FUNCTION_BLOCK Robot_Task_CAT (* Composite Function Block Type *)
  (* Standard: 61499-2 *)
  (* Version 0.0, 10/8/2025, Schneider Electric, template *)
  PACKAGE Main;
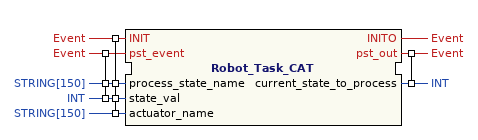
  EVENT_INPUT
    INIT WITH process_state_name, state_val, actuator_name; (* Initialization Request *)
    pst_event WITH process_state_name, state_val;
  END_EVENT
  EVENT_OUTPUT
    INITO; (* Initialization Confirm *)
    pst_out WITH current_state_to_process;
  END_EVENT
  VAR_INPUT
    process_state_name : STRING[150];
    state_val : INT;
    actuator_name : STRING[150];
  END_VAR
  VAR_OUTPUT
    current_state_to_process : INT;
  END_VAR
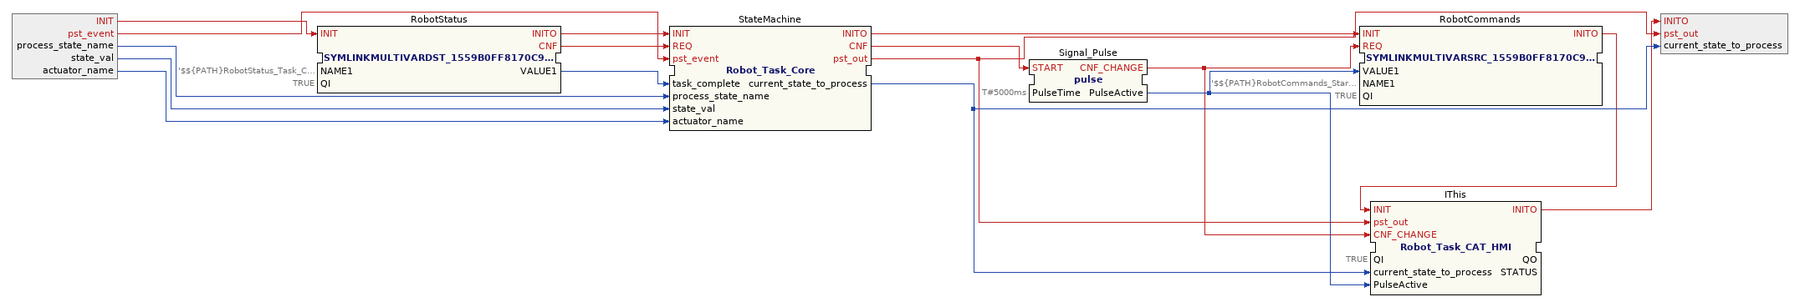
  FBS
    RobotCommands : SYMLINKMULTIVARSRC_1559B0FF8170C9BA0(NAME1 := '$${PATH}RobotCommands_StartTask', QI := TRUE); {SET_ATTRIBUTE(Configuration.GenericFBType.InterfaceParams, Runtime.System#I:=1;VALUE${I$}:BOOL)}
    RobotStatus : SYMLINKMULTIVARDST_1559B0FF8170C9BA0(NAME1 := '$${PATH}RobotStatus_Task_Complete', QI := TRUE); {SET_ATTRIBUTE(Configuration.GenericFBType.InterfaceParams, Runtime.System#I:=1;VALUE${I$}:BOOL)}
    StateMachine : Robot_Task_Core;
    Signal_Pulse : pulse(PulseTime := T#5000ms);
    IThis : Robot_Task_CAT_HMI(QI := TRUE);
  END_FBS
  EVENT_CONNECTIONS
    RobotStatus.INITO TO StateMachine.INIT;
    StateMachine.INITO TO RobotCommands.INIT;
    RobotStatus.CNF TO StateMachine.REQ;
    StateMachine.CNF TO Signal_Pulse.START;
    pst_event TO StateMachine.pst_event;
    StateMachine.pst_out TO pst_out;
    Signal_Pulse.CNF_CHANGE TO RobotCommands.REQ;
    INIT TO RobotStatus.INIT;
    RobotCommands.INITO TO IThis.INIT;
    StateMachine.pst_out TO IThis.pst_out;
    IThis.INITO TO INITO;
    Signal_Pulse.CNF_CHANGE TO IThis.CNF_CHANGE;
  END_CONNECTIONS
  DATA_CONNECTIONS
    RobotStatus.VALUE1 TO StateMachine.task_complete;
    StateMachine.current_state_to_process TO current_state_to_process;
    process_state_name TO StateMachine.process_state_name;
    state_val TO StateMachine.state_val;
    actuator_name TO StateMachine.actuator_name;
    Signal_Pulse.PulseActive TO RobotCommands.VALUE1;
    StateMachine.current_state_to_process TO IThis.current_state_to_process;
    Signal_Pulse.PulseActive TO IThis.PulseActive;
  END_CONNECTIONS
END_FUNCTION_BLOCK
